FUNCTION f_Addition : REAL
VAR_INPUT
	rSum1	:	REAL;
	rSum2	:	REAL;
END_VAR
VAR
END_VAR

f_Addition := rSum1 + rSum2;

END_FUNCTION

(* stored: Version 1.1.0.1, ProductVersion 3.1.4024.12
   POU f_Addition: Id {aca2f68e-fe14-40bb-b53a-9665046875f9}, SpecialFunc None *)
